# EPICS substitutions: iocs/testURRobot/iocBoot/ioctestURRobot/substitutions/canberra_13.substitutions
file "$(MCA)/mcaApp/Db/simple_mca.db"
{
pattern
{P           M       DTYP           INP         PREC  CHANS}
{testURRobot:med:   mca1  "asynMCA"   "@asyn(AIM2/1 0)"    3  2048}
{testURRobot:med:   mca2  "asynMCA"   "@asyn(AIM2/1 1)"    3  2048}
{testURRobot:med:   mca3  "asynMCA"   "@asyn(AIM2/1 2)"    3  2048}
{testURRobot:med:   mca4  "asynMCA"   "@asyn(AIM2/2 0)"    3  2048}
{testURRobot:med:   mca5  "asynMCA"   "@asyn(AIM2/2 1)"    3  2048}
{testURRobot:med:   mca6  "asynMCA"   "@asyn(AIM2/2 2)"    3  2048}
{testURRobot:med:   mca7  "asynMCA"   "@asyn(AIM3/1 0)"    3  2048}
{testURRobot:med:   mca8  "asynMCA"   "@asyn(AIM3/1 1)"    3  2048}
{testURRobot:med:   mca9  "asynMCA"   "@asyn(AIM3/1 2)"    3  2048}
{testURRobot:med:   mca10 "asynMCA"   "@asyn(AIM3/2 0)"    3  2048}
{testURRobot:med:   mca11 "asynMCA"   "@asyn(AIM3/3 1)"    3  2048}
{testURRobot:med:   mca12 "asynMCA"   "@asyn(AIM3/4 2)"    3  2048}
{testURRobot:med:   mca13 "asynMCA"   "@asyn(AIM3/2 3)"    3  2048}
{testURRobot:med:   mca0  "Soft Channel"   ""     3  2048}
}

file "$(MCA)/mcaApp/Db/icb_amp.db"
{
pattern
{P			AMP		PORT}
{testURRobot:med:	amp1	"icbAmp1"}
{testURRobot:med:	amp2	"icbAmp2"}
{testURRobot:med:	amp3	"icbAmp3"}
{testURRobot:med:	amp4	"icbAmp4"}
{testURRobot:med:	amp5	"icbAmp5"}
{testURRobot:med:	amp6	"icbAmp6"}
{testURRobot:med:	amp7	"icbAmp7"}
{testURRobot:med:	amp8	"icbAmp8"}
{testURRobot:med:	amp9	"icbAmp9"}
{testURRobot:med:	amp10	"icbAmp10"}
{testURRobot:med:	amp11	"icbAmp11"}
{testURRobot:med:	amp12	"icbAmp12"}
{testURRobot:med:	amp13	"icbAmp13"}
}

file "$(MCA)/mcaApp/Db/icb_adc.db"
{
pattern
{P			ADC		PORT}
{testURRobot:med:	adc1	"icbAdc1"}
{testURRobot:med:	adc2	"icbAdc2"}
{testURRobot:med:	adc3	"icbAdc3"}
{testURRobot:med:	adc4	"icbAdc4"}
}

file "$(MCA)/mcaApp/Db/icb_hvps.db"
{
pattern
{P			HVPS	LIMIT	PORT}
{testURRobot:med:	hvps1	1000	"icbHvps1"}
}
